FUNCTION_BLOCK FB_RobotMotion
VAR_INPUT
	iRunRoutine:BOOL; //TRUE to run the routine
	iRoutineNumber:INT; //target routine to run
	iTargetPosition:INT; //predicted  target positon to go to
	iInterlock:BOOL; //TRUE if is OK to go to target postion (pose)
	iTimeoutTime:TIME; //value for motion timeout
END_VAR

VAR_IN_OUT
	iqRobotData:structRobot;
	
END_VAR


VAR_OUTPUT
	qRoutineComplete: BOOL;
	qMotionTimeout: BOOL;
END_VAR
VAR
	timMotionTimeout: TON;
	// TRUE if the robot moved to a diffrent pose than was predicted
	qRoutinePoseFault: BOOL;
END_VAR
VAR // added by the converter: edge detectors and wires of the graphical bodies
    _rt1, _rt2, _rt3 : R_TRIG;
    _w1 : BOOL;
END_VAR

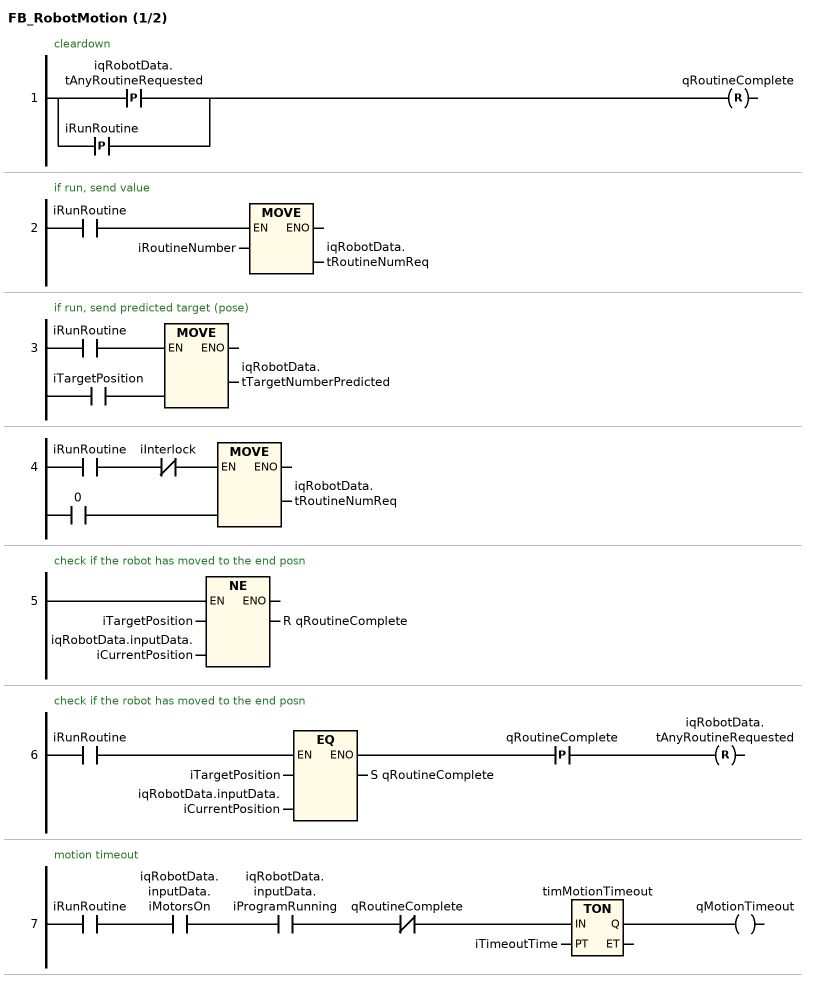
// NETWORK 1
// cleardown
_rt1(CLK := iqRobotData.tAnyRoutineRequested);
_rt2(CLK := iRunRoutine);
qRoutineComplete R= _rt1.Q OR _rt2.Q;

// NETWORK 2
// if run, send value
IF iRunRoutine THEN iqRobotData.tRoutineNumReq := iRoutineNumber; END_IF

// NETWORK 3
// if run, send predicted target (pose)
IF iRunRoutine THEN iqRobotData.tTargetNumberPredicted := iTargetPosition; END_IF

// NETWORK 4
IF iRunRoutine AND NOT iInterlock THEN iqRobotData.tRoutineNumReq := 0; END_IF

// NETWORK 5
// check if the robot has moved to the end posn
qRoutineComplete R= iTargetPosition <> iqRobotData.inputData.iCurrentPosition;

// NETWORK 6
// check if the robot has moved to the end posn
_w1 := iRunRoutine;
IF _w1 THEN qRoutineComplete S= iTargetPosition = iqRobotData.inputData.iCurrentPosition; END_IF
_rt3(CLK := qRoutineComplete);
iqRobotData.tAnyRoutineRequested R= _w1 AND _rt3.Q;

// NETWORK 7
// motion timeout
timMotionTimeout(IN := iRunRoutine AND iqRobotData.inputData.iMotorsOn AND iqRobotData.inputData.iProgramRunning AND NOT qRoutineComplete, PT := iTimeoutTime); // TON
qMotionTimeout := timMotionTimeout.Q;

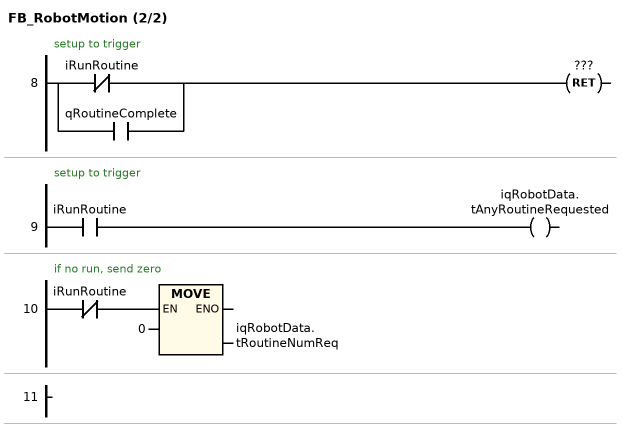
// NETWORK 8
// setup to trigger
IF NOT iRunRoutine OR qRoutineComplete THEN RETURN; END_IF

// NETWORK 9
// setup to trigger
iqRobotData.tAnyRoutineRequested := iRunRoutine;

// NETWORK 10
// if no run, send zero
IF NOT iRunRoutine THEN iqRobotData.tRoutineNumReq := 0; END_IF

// NETWORK 11

END_FUNCTION_BLOCK

(* stored: Version 1.1.0.1, ProductVersion 3.1.4024.11
   POU FB_RobotMotion: Id {8f4e82a4-e605-4e44-836b-9292c795164f}, SpecialFunc None *)
